FUNCTION_BLOCK T_CommandQueue EXTENDS T_NamedBase IMPLEMENTS I_CommandQueue
VAR
  low : T_TaskQueue;
  normal : T_TaskQueue;
  high : T_TaskQueue;
END_VAR
VAR CONSTANT
	BUFFERSIZE : UINT := 32;
END_VAR

METHOD AddHighPriority : BOOL
VAR_INPUT
  cmd : I_Task; 
END_VAR
AddHighPriority := AddWithPriority(cmd, E_CommandPriority.HIGH);
END_METHOD

METHOD AddLowPriority : BOOL
VAR_INPUT
  cmd : I_Task; 
END_VAR
AddLowPriority := AddWithPriority(cmd, E_CommandPriority.LOW);
END_METHOD

METHOD AddNormalPriority : BOOL
VAR_INPUT
  cmd : I_Task; 
END_VAR
AddNormalPriority := AddWithPriority(cmd, E_CommandPriority.NORMAL);
END_METHOD

METHOD AddWithPriority : BOOL
VAR_INPUT
  cmd : I_Task; 
  priority : E_CommandPriority;
END_VAR
VAR
  queueRef : REFERENCE TO T_TaskQueue;
END_VAR
IF cmd = 0 THEN
  LogError('Cant AddWithPriority() - cmd = 0 ');
  RETURN;
END_IF

IF Count >= BUFFERSIZE THEN
  LogError('Cant AddWithPriority() - Count >= BUFFERSIZE');
  RETURN;
END_IF

CASE priority OF
  E_CommandPriority.LOW:
    queueRef REF= low;
  E_CommandPriority.NORMAL:
    queueRef REF= normal;
  E_CommandPriority.HIGH:
    queueRef REF= high;
ELSE
  LogError(CONCAT('Unknown priority for command: ', TO_STRING(priority)));
  RETURN;

END_CASE

AddWithPriority := queueRef.Enqueue(cmd);

LogInfo(CONCAT(TO_STRING(priority),' priority command added to queue'));
END_METHOD

METHOD Clear
low.Clear();
normal.Clear();
high.Clear();

logInfo('Command queue cleared');
END_METHOD

PROPERTY Count : UINT
GET
//Combine all three queues and return the result
Count := Dint_to_Uint(high.Count + normal.Count + low.Count);
END_GET
END_PROPERTY

METHOD GetNext : BOOL
VAR_OUTPUT
	output_command : I_Task;
END_VAR
IF high.Count > 0 THEN
  IF high.TryDequeue(result => output_command) THEN
    LogInfo('High priority item dequeued');
    GetNext := TRUE;
    RETURN;

  ELSE
    GetNext := FALSE;
    RETURN;

  END_IF
ELSIF high.Count = 0 AND normal.Count > 0 THEN

  IF normal.TryDequeue(result => output_command) THEN
    LogInfo('Normal priority item dequeued');
    GetNext := TRUE;
    RETURN;

  ELSE
    GetNext := FALSE;
    RETURN;

  END_IF

ELSIF high.Count = 0 AND normal.Count = 0 AND low.Count > 0 THEN
  IF low.TryDequeue(result => output_command) THEN
    LogInfo('Low priority item dequeued');
    GetNext := TRUE;
    RETURN;

  ELSE
    GetNext := FALSE;
    RETURN;

  END_IF
END_IF
END_METHOD

END_FUNCTION_BLOCK

(* stored: Version 1.1.0.1
   POU T_CommandQueue: Id {5248d130-29dc-48c1-b42b-333676ef5f95}, SpecialFunc None
   Folder Methods: Id {ae58345e-57b5-4a0a-a056-6546bc7b39b3}
   Folder Properties: Id {030d4d2e-e25d-46c4-9ce5-65e25170095e}
   Method AddHighPriority: Id {71116a0c-490f-4af5-b5a8-a6907e7aa5f6}
   Method AddLowPriority: Id {3762e8f6-dc34-4f30-b13c-247c5171c1d4}
   Method AddNormalPriority: Id {61a64c53-93e9-4f81-b9b7-6c3d7147191f}
   Method AddWithPriority: Id {ea3bf24f-1aa3-4187-aba7-2c58cec368e6}
   Method Clear: Id {799a7323-5b88-490a-879a-0ce72518e31d}
   Property Count: Id {30c8b091-960f-48eb-a80e-7d1dcbebcc22}
   Get Get: Id {7fb86d84-c250-4512-8c94-b384361f4883}
   Method GetNext: Id {66b226ff-3080-42e8-a5cf-e1d5a467a42b} *)
